NETWORK
TITLE =KA: Handle commands
//Set the controlled stop and direct stop output signals.
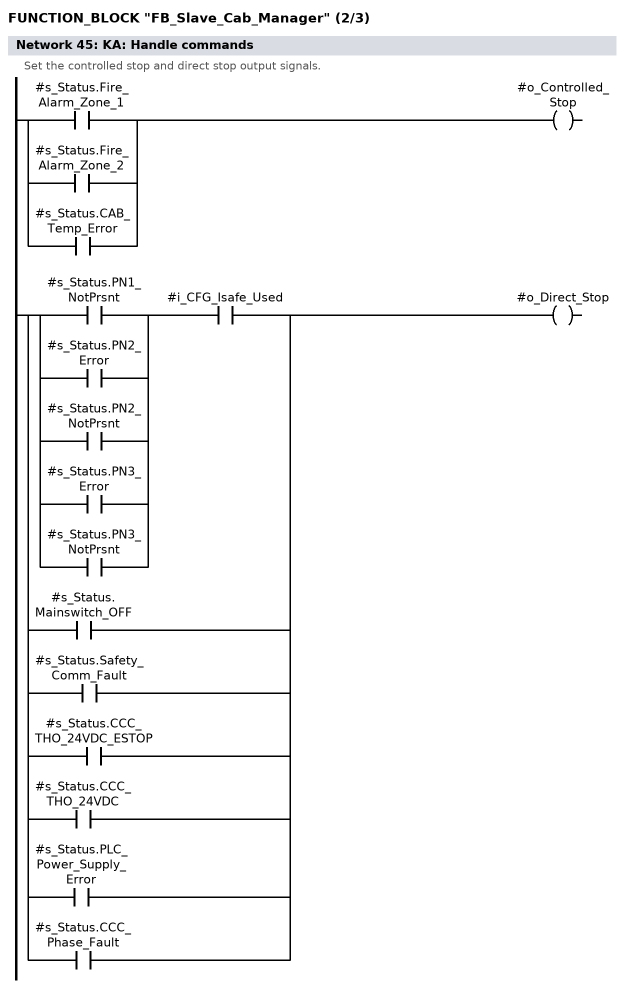
      O     #s_Status.Fire_Alarm_Zone_1;
      O     #s_Status.Fire_Alarm_Zone_2;
      O     #s_Status.CAB_Temp_Error;
      =     #o_Controlled_Stop;

      A(    ;
      O     #s_Status.PN1_NotPrsnt;
      O     #s_Status.PN2_Error;
      O     #s_Status.PN2_NotPrsnt;
      O     #s_Status.PN3_Error;
      O     #s_Status.PN3_NotPrsnt;
      )     ;
      A     #i_CFG_Isafe_Used;
      O     #s_Status.Mainswitch_OFF;
      O     #s_Status.Safety_Comm_Fault;
      O     #s_Status.CCC_THO_24VDC_ESTOP;
      O     #s_Status.CCC_THO_24VDC;
      O     #s_Status.PLC_Power_Supply_Error;
// Option to stop is Phase fault is detected.
      O     #s_Status.CCC_Phase_Fault;
      =     #o_Direct_Stop;
NETWORK
TITLE =LA: Write output signals
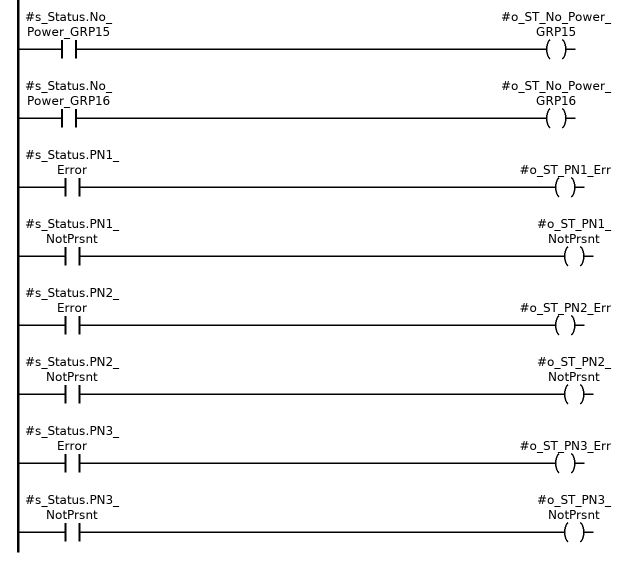

      A     #s_Status.Mainswitch_OFF;
      =     #o_ST_Mainswitch_OFF;

      A     #s_Status.Safety_Comm_Fault;
      =     #o_ST_Safety_Comm_Fault;

      A     #s_Status.CCC_THO_24VDC;
      =     #o_ST_CCC_THO_1_24VDC;

      A     #s_Status.PLC_Power_Supply_Error;
      =     #o_ST_CCC_THO_2_24VDC;

      A     #s_Status.CCC_THO_24VDC_ESTOP;
      =     #o_ST_CCC_THO_24VDC_ESTOP;

      A     #s_Status.CCC_THO_Phase;
      =     #o_ST_CCC_THO_Phase;

      A     #s_Status.CCC_Phase_Fault;
      =     #o_ST_CCC_Phase_Fault;

      A     #s_Status.Fire_Alarm_Zone_1;
      =     #o_ST_Fire_Alarm_Zone_1;

      A     #s_Status.Fire_Alarm_Zone_2;
      =     #o_ST_Fire_Alarm_Zone_2;

      A     #s_Status.ETH_Switch_Fault;
      =     #o_ST_ETH_Switch_Fault;

      A     #s_Status.CAB_Temp_High;
      =     #o_ST_CAB_Temp_Error;

      A     #s_Status.CAB_Temp_Error;
      =     #o_ST_CAB_Temp_Error;

      A     #s_Status.UPS_THO;
      =     #o_ST_UPS_THO;

      A     #s_Status.THO_400VAC_GRP01;
      =     #o_ST_THO_400Vac_GRP01;

      A     #s_Status.THO_400VAC_GRP02;
      =     #o_ST_THO_400Vac_GRP02;

      A     #s_Status.THO_400VAC_GRP03;
      =     #o_ST_THO_400Vac_GRP03;

      A     #s_Status.THO_400VAC_GRP04;
      =     #o_ST_THO_400Vac_GRP04;

      A     #s_Status.THO_400VAC_GRP05;
      =     #o_ST_THO_400Vac_GRP05;

      A     #s_Status.THO_400VAC_GRP06;
      =     #o_ST_THO_400Vac_GRP06;

      A     #s_Status.THO_400VAC_GRP07;
      =     #o_ST_THO_400Vac_GRP07;

      A     #s_Status.THO_400VAC_GRP08;
      =     #o_ST_THO_400Vac_GRP08;

      A     #s_Status.THO_400VAC_GRP09;
      =     #o_ST_THO_400Vac_GRP09;

      A     #s_Status.THO_400VAC_GRP10;
      =     #o_ST_THO_400Vac_GRP10;

      A     #s_Status.THO_400VAC_GRP11;
      =     #o_ST_THO_400Vac_GRP11;

      A     #s_Status.THO_400VAC_GRP12;
      =     #o_ST_THO_400Vac_GRP12;

      A     #s_Status.THO_400VAC_GRP13;
      =     #o_ST_THO_400Vac_GRP13;

      A     #s_Status.THO_400VAC_GRP14;
      =     #o_ST_THO_400Vac_GRP14;

      A     #s_Status.THO_400VAC_GRP15;
      =     #o_ST_THO_400Vac_GRP15;

      A     #s_Status.THO_400VAC_GRP16;
      =     #o_ST_THO_400Vac_GRP16;

      A     #s_Status.THO_230VAC_GRP01;
      =     #o_ST_THO_230Vac_GRP01;

      A     #s_Status.THO_230VAC_GRP02;
      =     #o_ST_THO_230Vac_GRP02;

      A     #s_Status.THO_230VAC_GRP03;
      =     #o_ST_THO_230Vac_GRP03;

      A     #s_Status.THO_230VAC_GRP04;
      =     #o_ST_THO_230Vac_GRP04;

      A     #s_Status.THO_230VAC_GRP05;
      =     #o_ST_THO_230Vac_GRP05;

      A     #s_Status.THO_230VAC_GRP06;
      =     #o_ST_THO_230Vac_GRP06;

      A     #s_Status.THO_230VAC_GRP07;
      =     #o_ST_THO_230Vac_GRP07;

      A     #s_Status.THO_230VAC_GRP08;
      =     #o_ST_THO_230Vac_GRP08;

      A     #s_Status.THO_230VAC_GRP09;
      =     #o_ST_THO_230Vac_GRP09;

      A     #s_Status.THO_230VAC_GRP10;
      =     #o_ST_THO_230Vac_GRP10;

      A     #s_Status.THO_230VAC_GRP11;
      =     #o_ST_THO_230Vac_GRP11;

      A     #s_Status.THO_230VAC_GRP12;
      =     #o_ST_THO_230Vac_GRP12;

      A     #s_Status.THO_230VAC_GRP13;
      =     #o_ST_THO_230Vac_GRP13;

      A     #s_Status.THO_230VAC_GRP14;
      =     #o_ST_THO_230Vac_GRP14;

      A     #s_Status.THO_230VAC_GRP15;
      =     #o_ST_THO_230Vac_GRP15;

      A     #s_Status.THO_230VAC_GRP16;
      =     #o_ST_THO_230Vac_GRP16;

      A     #s_Status.No_Power_GRP01;
      =     #o_ST_No_Power_GRP01;

      A     #s_Status.No_Power_GRP02;
      =     #o_ST_No_Power_GRP02;

      A     #s_Status.No_Power_GRP03;
      =     #o_ST_No_Power_GRP03;

      A     #s_Status.No_Power_GRP04;
      =     #o_ST_No_Power_GRP04;

      A     #s_Status.No_Power_GRP05;
      =     #o_ST_No_Power_GRP05;

      A     #s_Status.No_Power_GRP06;
      =     #o_ST_No_Power_GRP06;

      A     #s_Status.No_Power_GRP07;
      =     #o_ST_No_Power_GRP07;

      A     #s_Status.No_Power_GRP08;
      =     #o_ST_No_Power_GRP08;

      A     #s_Status.No_Power_GRP09;
      =     #o_ST_No_Power_GRP09;

      A     #s_Status.No_Power_GRP10;
      =     #o_ST_No_Power_GRP10;

      A     #s_Status.No_Power_GRP11;
      =     #o_ST_No_Power_GRP11;

      A     #s_Status.No_Power_GRP12;
      =     #o_ST_No_Power_GRP12;

      A     #s_Status.No_Power_GRP13;
      =     #o_ST_No_Power_GRP13;

      A     #s_Status.No_Power_GRP14;
      =     #o_ST_No_Power_GRP14;

      A     #s_Status.No_Power_GRP15;
      =     #o_ST_No_Power_GRP15;

      A     #s_Status.No_Power_GRP16;
      =     #o_ST_No_Power_GRP16;

      A     #s_Status.PN1_Error;
      =     #o_ST_PN1_Err;

      A     #s_Status.PN1_NotPrsnt;
      =     #o_ST_PN1_NotPrsnt;

      A     #s_Status.PN2_Error;
      =     #o_ST_PN2_Err;

      A     #s_Status.PN2_NotPrsnt;
      =     #o_ST_PN2_NotPrsnt;

      A     #s_Status.PN3_Error;
      =     #o_ST_PN3_Err;

      A     #s_Status.PN3_NotPrsnt;
      =     #o_ST_PN3_NotPrsnt;

END_FUNCTION_BLOCK

